FUNCTION_BLOCK BASIC_STORAGE_DINT (* Basic Function Block Type *)
  (* Standard: 61499-2 *)
  (* Version 0.0, 4/30/2023, Dmitrii, Flexbridge AB, Template *)
  PACKAGE UAO.Hackathon;
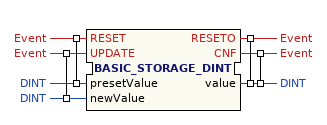
  EVENT_INPUT
    RESET WITH presetValue; (* Reset output to presetValue *)
    UPDATE WITH newValue; (* Set output value to newValue *)
  END_EVENT
  EVENT_OUTPUT
    RESETO WITH value; (* Reset confirnmation *)
    CNF WITH value; (* Execution Confirmation *)
  END_EVENT
  VAR_INPUT
    presetValue : DINT; (* Reset value *)
    newValue : DINT; (* New value to capture on UPDATE *)
  END_VAR
  VAR_OUTPUT
    value : DINT; (* Output value *)
  END_VAR
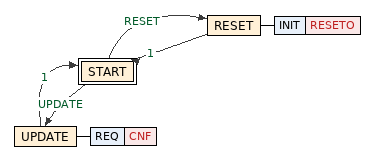
  EC_STATES
    START; (* Initial State *)
    RESET : INIT -> RESETO; (* Initialization *)
    UPDATE : REQ -> CNF; (* Normal execution *)
  END_STATES
  EC_TRANSITIONS
    START TO RESET := RESET;
    RESET TO START := 1;
    START TO UPDATE := UPDATE;
    UPDATE TO START := 1;
  END_TRANSITIONS
  ALGORITHM INIT IN ST: (* Initialization algorithm *)
;
value:=presetValue;
  END_ALGORITHM
  ALGORITHM REQ IN ST: (* Normally executed algorithm *)
;
value:=newValue;
  END_ALGORITHM
END_FUNCTION_BLOCK
